(*======================================================================================================================================*)
(*//=============================================================================\\
||  _   _ _  __  _         _                        _   _                      ||
|| | \ | | |/ / / \  _   _| |_ ___  _ __ ___   __ _| |_(_) ___  _ __         ||
|| |  \| | ' / / _ \| | | | __/ _ \| '_ ` _ \ / _` | __| |/ _ \| '_ \        ||
|| | |\  | . \/ ___ \ |_| | || (_) | | | | | | (_| | |_| | (_) | | | |       ||
|| |_| \_|_|\_\_/  \_\__,_|\__\___/|_| |_| |_|\__,_|\__|_|\___/|_| |_|       ||
||                                                                             ||
\\=============================================================================//
fb_RS485FiFoMaster:	Einfaches Senden eines Telegrams über RS485*)
(*
Date          	| Version    	| created under        	| Author          	| Remark *)
(*====================================================================================================================================================*)
(*10/05/2025   	| 1.00      		| TC3		  		| N.Kersting       | first release *)
(*10/05/2025   	| 1.01      		| TC3		  		| N.Kersting       | Nun wird der Empfang auch mit Implementiert  *)
(*13/05/2025   	| 1.02      		| TC3		  		| N.Kersting       | Busbelastungstest Implementiert - Sendet Durchgehend Strings *)
(*14/05/2025   	| 1.03      		| TC3		  		| N.Kersting       | Busauslastung direkt Implementiert *)
(*27/05/2025   	| 1.04      		| TC3		  		| N.Kersting       | Neuen Manuell Mode implementiert um einen Manuell generierten String allein zu Senden *)
(*28/05/2025   	| 1.05      		| TC3		  		| N.Kersting       | Neue Automatisch Ping Funktion hinzugefügt & Wichtiger Bugfix *)
(*02/06/2025   	| 2.00      		| TC3		  		| N.Kersting       | Neue Verbesserte Collision Detection, verhindert, dass Senden bei gefülltem Epmfangspuffer *)
(*03/06/2025   	| 2.01      		| TC3		  		| N.Kersting       | Collision Detection nun aufgeeilt in Empfang und Senden *)
(*03/06/2025   	| 2.02      		| TC3		  		| N.Kersting       | Neue Bus Scan Funktion Implementiert, Scannt alle Teilnehmer Ids im Bus (nur im Manuell Mode verfügbar) *)
(*12/01/2026   	| 2.03      		| TC3		  		| N.Kersting       | Nach dem Pingenkann wieder empfangen werden*)
(*13/01/2026   	| 2.04      		| TC3		  		| N.Kersting       | Ping wird Verzögert zwischen jedem Ping, wenn FiFo gefüllt kann Ping unterbrochen werden*)
(*13/01/2026   	| 2.04      		| TC3		  		| N.Kersting       | Bugfix Step 12 nur speichern wenn ID vorhanden ist!*)
(*09/06/2026   	| 2.05      		| TC3		  		| N.Kersting       | Obergrenze für Max Rows FiFo nun fix auf Globalen Wert *)
(*09/06/2026   	| 2.06      		| TC3		  		| N.Kersting       | Integration I_nMaxDevices*)
(*16/09/2026   	| 2.07      		| TC3		  		| N.Kersting       | Collision Detection eingang*)
(*====================================================================================================================================================*)
FUNCTION_BLOCK fb_RS485FiFoMaster_old
VAR_INPUT
	I_nMaxDevices				:INT := cMaxRowCMDFiFo;
	I_sSendCmdFiFo				:ARRAY[1..cMaxRowCMDFiFo] OF STRING(255);
	I_stDeviceIdent				:ARRAY[1..cMaxRowCMDFiFo] OF ST_HausBus_Ident;	(* Um Zyklisch einzelnt anzupingen *)
	
	I_bAutoPing					:BOOL;												(* Wenn Aktiv wird Zyklisch Automatisch ein Ping gesendet, welcher von den einzelnen Kommunikationsbausteinen ausgewertet werden kann *)
	I_tAutoPingTime				:TIME :=T#10S;										(* Die Intervallzeit, Bis ein Auto Ping gesendet wird *)
	
	I_bUseRXCollisionDetection	:BOOL := TRUE;					(* Aktiviert die Empfangs Kollisions Überprüfung *)
	I_bUseTXCollisionDetection	:BOOL := FALSE;					(* Aktiviert die Sende Kollisions Überprüfung *)
	I_tVerzCollisionDetect		:TIME := T#100MS;
	
	I_bManuellMode				:BOOL := FALSE;
	I_bSearchMode				:BOOL := FALSE;
	I_sSendCmdManuell			:STRING(255);
	I_bSendManuell				:BOOL;
	I_bLogger					:BOOL := FALSE;
	I_bResetLog					:BOOL := FALSE;
	I_bExecute					:BOOL := TRUE;
	I_bBusBelastungstest		:BOOL;
	I_bReset					:BOOL;
	I_sStartZeichen				:BYTE := 16#FD;										(* Startzeichen Präfix *)
	I_sEndZeichen				:BYTE := 16#FE;										(* Endzeichen Suffix *)
	I_pTxBuffer					:POINTER TO ComBuffer; 								(* Zeiger auf TX-Buffer*)
	I_pRxBuffer   				:POINTER TO ComBuffer;  							(* Zeiger auf RX-Buffer*)
END_VAR
VAR_OUTPUT
	Q_bSendDoneFiFo				:ARRAY[1..cMaxRowCMDFiFo] OF BOOL; (*GVL_RS485FiFoSend.bSendDoneFiFo[iFiFoRow]*)
	Q_sReceiveString			:STRING(255);		
	Q_lrBusAuslastung			:LREAL;
	Q_bBusy						:BOOL;
	Q_bDone						:BOOL;
	Q_bError					:BOOL;
	Q_sState					:STRING;
	Q_stStates					:ST_FiFoMaster_State;
END_VAR
VAR
(*==========================================================================================================*)
(* Parameter *)
(*==========================================================================================================*)
	bActivateSend				:BOOL := TRUE;					(* Aktiviert das Senden von Nachrichten *)
	bActivateReceive			:BOOL := TRUE;					(* Aktiviert das Empfangen von Nachrichten *)
	
	bUseRXCollisionDetection	:BOOL := TRUE;					(* Aktiviert die Empfangs Kollisions Überprüfung *)
	bUseTXCollisionDetection	:BOOL := FALSE;					(* Aktiviert die Sende Kollisions Überprüfung *)
	tVerzCollisionDetect		:TIME := T#100MS;				(* Zeit, die zum Empfangen bleibt *)
(*==========================================================================================================*)	
	bRXCollisionDetected		:BOOL;
	bTXCollisionDetected		:BOOL;
	bCollisionFree				:BOOL;	
(*==========================================================================================================*)		
	bFirstCycle					:BOOL := TRUE;
	bStringSend					:BOOL := FALSE;
	bBusBelastungstest			:BOOL := FALSE;
	bBusAuslastung				:BOOL := TRUE;
	bPingStart					:BOOL;
	bBusyMem					:BOOL;
(*==========================================================================================================*)	
	sReceivedMEMString			:STRING(255);
	sReceivedString				:STRING(255);
	sStep						:STRING;
	sString						:STRING(255);
	sStringSend					:STRING(255);
(*==========================================================================================================*)		
	iStep						:INT;
	iStepReceive				:INT;
	iMaxBufferBlocking			:INT := 20;
	icntError					:INT;
	iFiFoRow					:INT := 1;
	icntFiFo					:INT;
	i,h							:INT;
	iStepFiFo					:INT;
	iPingRow					:INT;
(*==========================================================================================================*)		

	tonCollisionFree			:ton;	
	tonTimeout					:ton;
	tonPingIntervall			:ton;
	tonPingVerz					:ton;
	tonSend						:ton;
(*==========================================================================================================*)		
	rTrigSendManuell			:r_Trig;
	rTrigSendSearchMode			:r_trig;
	fbSend     					:SendString255;
	fbReceive   				:ReceiveString255;
	
	fbBusAuslastung				:fb_FilterArray;
	
	fbRS485Search				:fb_RS485IdScan;
	
	fbRS485Logger				:fb_RS485Logger;
	
END_VAR

(*============================================================================================*)
(* Laufzeit fehler *)
tonTimeout(
	PT:=T#1S);
	
(*============================================================================================*)		
(* Collision detection, soll verhinddern, dass nicht gesendet wird, wenn Daten im Empfangsüpuffer sind *)
bUseRXCollisionDetection := I_bUseRXCollisionDetection;
bUseTXCollisionDetection := I_bUseTXCollisionDetection;

(* Receive Collision Dectetion *)
bRXCollisionDetected :=	(I_pRxBuffer^.Count > INT_TO_UINT(iMaxBufferBlocking) 
						OR I_pRxBuffer^.FreeByte < (301 -INT_TO_UINT(iMaxBufferBlocking))
						OR I_pRxBuffer^.blocked
						OR I_pRxBuffer^.Error <> 0
						OR fbReceive.StringReceived
						(*OR sReceivedString <> ''*))
						AND bUseRXCollisionDetection;
						
(* Transmit Collision Detection *)
bTXCollisionDetected :=	(I_pTxBuffer^.Count > INT_TO_UINT(iMaxBufferBlocking) 
						OR I_pTxBuffer^.FreeByte < (301 -INT_TO_UINT(iMaxBufferBlocking))
						OR I_pTxBuffer^.blocked
						OR I_pTxBuffer^.Error <> 0)
						AND bUseTXCollisionDetection;
						
(* Collision Detection Verzögern *)	
tVerzCollisionDetect :=		I_tVerzCollisionDetect;
			
tonCollisionFree(
	IN := 	NOT bRXCollisionDetected
			AND NOT bTXCollisionDetected,
	PT := 	tVerzCollisionDetect,
	Q =>	bCollisionFree);

(*============================================================================================*)	
(* Ping Intervall Timer *)		
tonPingIntervall(
	IN := I_bAutoPing
			AND NOT bPingStart,
	PT := I_tAutoPingTime);

tonPingVerz(
	PT := T#100MS);	
	
(*============================================================================================*)	
(* Busbelastungstest *)	
bBusBelastungstest := I_bBusBelastungstest;
sReceivedMEMString:='';

(*============================================================================================*)	
(* Anzahl der gefüllten FiFo Zeilen *)
icntFiFo := 0;
FOR i := 1 TO cMaxRowCMDFiFo BY 1 DO 
	
	IF i <= I_nMaxDevices
	THEN
		IF (I_sSendCmdFiFo[i]<> '')
		THEN
			icntFiFo := icntFiFo +1;
		END_IF
	END_IF
END_FOR

(*============================================================================================*)	
(* Manuelles Senden *)
rTrigSendManuell(
	CLK := I_bSendManuell);

(*============================================================================================*)
CASE iStepFiFo OF
-1:	sStep := 'FiFo INIT';
	bFirstCycle := FALSE;
	Q_bBusy := FALSE;
	bPingStart := FALSE;
	iFiFoRow := 1;
	iPingRow := 1;
	
	FOR h := 1 TO cMaxRowCMDFiFo BY 1 DO
		IF h <= I_nMaxDevices
		THEN
			Q_bSendDoneFiFo[h] :=TRUE;
		END_IF
	END_FOR
	
	iStepFiFo := 0;

(*============================================================================================*)
0:	sStep := 'Warten, dass FiFo gefüllt wird';
	iFiFoRow := 1;
	
	IF iPingRow <= 0
	THEN
		iPingRow := 1;
	END_IF
	
	bStringSend := FALSE;
	Q_bBusy := FALSE;
	tonPingVerz.IN := FALSE;
		
	(* Wenn die Intervall Zeit abgelaufen ist Ping Start setzen *)
	IF tonPingIntervall.Q
	THEN
		bPingStart := TRUE;
	END_IF
	
	(*IF (icntFiFo > 0
		OR  bBusBelastungstest
		OR I_bManuellMode)
		AND NOT bFirstCycle
		AND NOT bPingStart
		AND bCollisionFree
	THEN
		Q_bBusy := TRUE;
		iStepFiFo := 1;
	ELSIF
		bFirstCycle
	THEN
		iStepFiFo := -1;
	ELSIF
	(* (	*)(bPingStart
		AND NOT bFirstCycle)
		(*OR (bPingStart
		AND iPingRow <> cMaxRS485CMDFiFo))*) (* Es stehen noch Ping befehle aus *)
		AND bCollisionFree
		(*AND icntFiFo =0*)
	THEN
		(*iFiFoRow := iPingRow;*)
		iStepFiFo := 10;	(* Ping senden *)
	END_IF*)
	
	IF bFirstCycle
	THEN
		iStepFiFo := -1;
	ELSE
		IF bCollisionFree
		THEN
			IF icntFiFo > 0
				OR  bBusBelastungstest
				OR I_bManuellMode
			THEN
				Q_bBusy := TRUE;
				iStepFiFo := 1;
			ELSE
				IF bPingStart
					OR iPingRow < I_nMaxDevices	(* Ping wurde unterbrochen *)
				THEN
					IF iPingRow < I_nMaxDevices
					THEN
						iFiFoRow := iPingRow;
					ELSE
						iFiFoRow := 1;
					END_IF
					iStepFiFo := 10;	(* Ping senden *)
				END_IF
			END_IF
		END_IF
	END_IF
	
(*============================================================================================*)	
1:	sStep := 'Prüfen ob STRING in FiFo Zeile gefüllt*';
	
	IF I_bSearchMode
	THEN
		sStep :=fbRS485Search.Q_sState;
	END_IF
	
	(* Manueller Modus *)
	IF I_bManuellMode
	THEN
		(* Prüfen ob in der Zeile etwas steht *)
		IF I_sSendCmdManuell <>''
			AND rTrigSendManuell.Q
			AND NOT I_bSearchMode
		THEN
			IF bCollisionFree
			THEN
				sString :=	I_sSendCmdManuell; 
				bStringSend := TRUE;
				Q_bDone := FALSE;
				Q_bError := FALSE;
				iStepFiFo := iStepFiFo+1;
			END_IF
		END_IF
		(* Prüfen ob in der Zeile etwas steht *)
		IF I_bSearchMode
			AND fbRS485Search.Q_bSend
		THEN
			IF bCollisionFree
			THEN
				sString :=	fbRS485Search.Q_sSearchString; 
				bStringSend := TRUE;
				Q_bDone := FALSE;
				Q_bError := FALSE;
				iStepFiFo := iStepFiFo+1;
			END_IF
		END_IF
	ELSE
		(* Prüfen ob in der ausgewählten Zeile etwas steht *)
		sStringSend :=	I_sSendCmdFiFo[iFiFoRow]; 
		IF I_sSendCmdFiFo[iFiFoRow] = ''
		THEN
			IF iFiFoRow< I_nMaxDevices
			THEN
				iFiFoRow := iFiFoRow+1; (* Nächste Zeile, bis etwas drin Steht *)
			ELSE
				IF bBusBelastungstest
				THEN
					sStringSend :=	CONCAT(F_ToCHR(I_sStartZeichen),'ServiceTOOL-BUSBELASTUNGSTEST-BURSTFIREMODE');
					sStringSend :=	CONCAT(sStringSend,F_ToCHR(I_sEndZeichen));
					(* Senden *)
					
					IF  bCollisionFree
					THEN
						sStep := 'Prüfe ob Senden noch aktiv ist';
						bStringSend := TRUE;
						sString :=	sStringSend;
						Q_bDone := FALSE;
						Q_bError := FALSE;
						iStepFiFo := iStepFiFo+1;
					END_IF
				ELSE
					iStepFiFo := 0;	(* Alle Zeilen Abgearbeitet *)
				END_IF
			END_IF
		ELSE
		(* Senden *)
		Q_bSendDoneFiFo[iFiFoRow] :=FALSE;
		
			IF bCollisionFree
			THEN
				sStep := 'Prüfe ob Senden noch aktiv ist';
				bStringSend := TRUE;
				sString :=	sStringSend;
				Q_bDone := FALSE;
				Q_bError := FALSE;
				iStepFiFo := iStepFiFo+1;
			END_IF
		END_IF
	END_IF
	
(*============================================================================================*)		
2:	sStep := 'Starte Senden';
	Q_bBusy := TRUE;
	tonTimeout.IN := fbSend.Busy;
	
	IF NOT fbSend.Busy
		AND NOT fbReceive.StringReceived
	THEN
		sString := '';
		tonSend.IN := FALSE;
		bStringSend := FALSE;
		iStepFiFo := iStepFiFo+1;
	ELSIF
		(fbSend.Error >0)
		AND NOT (fbSend.Error = 2)
	THEN
		sStep := CONCAT('ERROR-',sStep);
		sStep := CONCAT(sStep,'- ');
		sStep := CONCAT(sStep,INT_TO_STRING(fbSend.Error));
		iStepFiFo := -2;
	ELSIF
		tonTimeout.Q
	THEN
		sStep := CONCAT('ERROR- Timeout',sStep);
		iStepFiFo := -2;
	END_IF
	
(*============================================================================================*)		
3:	(* Senden*)		
	Q_bSendDoneFiFo[iFiFoRow] :=TRUE;
	
	IF iFiFoRow< I_nMaxDevices
		AND NOT I_bSearchMode
	THEN
		iFiFoRow := iFiFoRow+1;
		iStepFiFo := 1;
	ELSE
		Q_bDone := TRUE;
		
		IF (NOT fbRS485Search.Q_bSend
			AND I_bSearchMode)
			OR NOT I_bSearchMode
		THEN
			iStepFiFo := 0;
		END_IF
		
	END_IF
	
(*============================================================================================*)	
(* Ping Senden Ablauf *)
(*============================================================================================*)	
10:	sStep := 'Sende Ping*';
	
	tonPingVerz.IN := FALSE;
	
	(* Ping String erstellen *)
	sStringSend:=	CONCAT(F_ToCHR(I_sStartZeichen),DINT_TO_STRING(I_stDeviceIdent[iFiFoRow].diID));
	sStringSend :=	CONCAT(sStringSend,'.');
	sStringSend :=	CONCAT(sStringSend ,I_stDeviceIdent[iFiFoRow].sPingIdent); 
	sStringSend :=	CONCAT(sStringSend,F_ToCHR(I_sEndZeichen));
	
	IF I_stDeviceIdent[iFiFoRow].sPingIdent = ''
		OR I_stDeviceIdent[iFiFoRow].diID = 0
	THEN
		IF iFiFoRow < I_nMaxDevices
		THEN
			iFiFoRow := iFiFoRow+1; (* Nächste Zeile, bis etwas drin Steht *)
		ELSE
			bPingStart := FALSE;
			iPingRow := I_nMaxDevices;
			iStepFiFo := 0;	(* Alle Zeilen Abgearbeitet *)
		END_IF
	ELSE
	(* Senden *)	
		IF bCollisionFree
		THEN
			sStep := 'Prüfe ob Senden noch aktiv ist';
			bStringSend := TRUE;
			sString :=	sStringSend;
			Q_bDone := FALSE;
			Q_bError := FALSE;
			iStepFiFo := iStepFiFo+1;
		END_IF
	END_IF
	
(*============================================================================================*)		
11:	sStep := 'Starte Senden';
	Q_bBusy := TRUE;
	tonTimeout.IN := fbSend.Busy;
	
	IF NOT fbSend.Busy
		(*AND NOT fbReceive.StringReceived*)
	THEN
		tonSend.IN := FALSE;
		bStringSend := FALSE;
				
		IF NOT fbReceive.StringReceived
			AND bCollisionFree
		THEN
			iStepFiFo := iStepFiFo+1;
		END_IF
		
	ELSIF
		(fbSend.Error >0)
		AND NOT (fbSend.Error = 2)
	THEN
		sStep := CONCAT('ERROR-',sStep);
		sStep := CONCAT(sStep,'- ');
		sStep := CONCAT(sStep,INT_TO_STRING(fbSend.Error));
		iStepFiFo := -2;
	ELSIF
		tonTimeout.Q
	THEN
		sStep := CONCAT('ERROR- Timeout',sStep);
		iStepFiFo := -2;
	END_IF
	
(*============================================================================================*)		
12:	(* Senden*)		
	(* Nur speichern wenn auch wirklich eine ID vorhanden ist *)	
	IF I_stDeviceIdent[iFiFoRow].sPingIdent = ''
		OR I_stDeviceIdent[iFiFoRow].diID = 0
	THEN
		IF iFiFoRow < I_nMaxDevices
		THEN
			iFiFoRow := iFiFoRow+1; (* Nächste Zeile, bis etwas drin Steht *)
		ELSE
			bPingStart := FALSE;
			iPingRow := I_nMaxDevices;
			iStepFiFo := 0;	(* Alle Zeilen Abgearbeitet *)
		END_IF
	ELSE
		IF iFiFoRow < I_nMaxDevices
		THEN
			iFiFoRow := iFiFoRow+1;
			iPingRow := iFiFoRow; (* Zeile speichern *)
			iStepFiFo := 13;	(* Falls das warten Deaktiviert werden soll, kann hier einfach in 10 gesprungen werden *)
		ELSE
			bPingStart := FALSE; (* Letzte Ping Zeile erreicht, Timer zurücksetzen  *)
			iPingRow := I_nMaxDevices;
			iStepFiFo := 13;
		END_IF
	END_IF
(*============================================================================================*)		
13:	(* Optionale Wartezeit zwischen jedem Ping*)		
	tonPingVerz.IN := TRUE;
			
	IF tonPingVerz.Q
	THEN
		IF NOT fbReceive.StringReceived
			AND bCollisionFree
		THEN
			tonPingVerz.IN := FALSE;
			
			IF iFiFoRow < I_nMaxDevices
			THEN
				iStepFiFo := 10; (* nächsten Ping senden *)
			ELSE
				iStepFiFo := 0;
			END_IF
		END_IF
	ELSE
		(* Prüfen ob ein Sendeauftrag anliegt *)
		IF icntFiFo >0
		THEN
			tonPingVerz.IN := FALSE;
			iStepFiFo := 0; (* Sende FiFo leeren *)
		END_IF  
	END_IF
ELSE
(*============================================================================================*)
	Q_bError := TRUE;
	Q_bBusy := FALSE;
	bBusyMem := FALSE;
	tonTimeout.IN := FALSE;
	
	IF I_bReset
	THEN
		iStepFiFo := 0;
	END_IF
END_CASE

(*============================================================================================*)	
(* Nur Senden, wenn nicht Empfangen wird *)
IF bStringSend
THEN
	IF bActivateSend
	THEN
		(* Senden *)
		fbSend(
			SendString:= 	sString,
			TXbuffer:= 		I_pTxBuffer^);
	END_IF
	
ELSE
	IF bActivateReceive
	THEN
		(* Empfangen *)
		ac00_Receive();
	END_IF
END_IF

(*============================================================================================*)	
(* Empfangsmerker 0 Setzen am ende Eines Zyklus *)
Q_sReceiveString := sReceivedMEMString;

(*============================================================================================*)	
(* Busauslastung tracken*)
ac99_Diagnose();

(*============================================================================================*)	
(* StatusStruktur für Visu *)
Q_sState :=	sStep;
Q_stStates.bBusy				:=	Q_bBusy;
Q_stStates.bDone				:=	Q_bDone;
Q_stStates.bError				:=	Q_bError;
Q_stStates.iFiFoCount			:=	icntFiFo;
Q_stStates.iFiFoRow				:=	iFiFoRow;
Q_stStates.lrBusAuslastung		:=	Q_lrBusAuslastung;
Q_stStates.sReceiveString 		:=	Q_sReceiveString;
Q_stStates.sSendString 			:=	sString;
Q_stStates.sState 				:=	Q_sState;

(*============================================================================================*)	
(* RS485 Telegramm Logging *)
fbRS485Logger(
	I_bExecute:= 		I_bLogger,						(* oder eine externe Variable *)
	I_bReset:=			I_bResetLog,	
	I_sTxTelegram:= 	sString,
	I_sRxTelegram:= 	sReceivedMEMString);

ACTION ac00_Receive:
(*============================================================================================*)	
(* Empfangen *)

CASE iStepReceive OF		
0:	fbReceive(
		Prefix := 			F_ToCHR(I_sStartZeichen),
		Suffix := 			F_ToCHR(I_sEndZeichen),
		Timeout:= , 
		Reset:= , 
		StringReceived=> , 
		Busy=> , 
		Error=> , 
		RxTimeout=> , 
		ReceivedString:= 	sReceivedString, 
		RXbuffer:= 			I_pRxBuffer^);
		
	IF fbReceive.StringReceived
	THEN
		iStepReceive := 1;
		sReceivedMEMString := sReceivedString;
	END_IF
	
1:	sReceivedString := '';
	iStepReceive := 0;

	
END_CASE
END_ACTION

ACTION ac99_Diagnose:
(*============================================================================================*)	
(* Busauslastung Prüfen *)

fbBusAuslastung(
	I_bExcecute:= 	bBusAuslastung, 
	I_nWert:= 		UINT_TO_LREAL(I_pTxBuffer^.Count), 
	I_nFilterWert:= 50, 
	Q_nFilter=> 	Q_lrBusAuslastung);
	
	
fbRS485Search(
	I_bStartSearch:= 	I_bSearchMode, 
	I_diStartID:= , 
	I_diMaxID:= , 
	I_sStartZeichen:= 	I_sStartZeichen, 
	I_sEndZeichen:= 	I_sEndZeichen, 
	I_tWait:= , 
	I_StringReceived:= 	sReceivedMEMString, 
	Q_bSend=> , 
	Q_sSearchString=> );
END_ACTION

END_FUNCTION_BLOCK

(* stored: Version 1.1.0.1, ProductVersion 3.1.4024.16
   POU fb_RS485FiFoMaster_old: Id {abb7ee14-f2e6-4645-9657-7cebd7b41d33}, SpecialFunc None
   Action ac00_Receive: Id {c12285ff-9b41-4e09-9783-e6434850ec65}
   Action ac99_Diagnose: Id {729e27f4-8df9-41ab-a478-b2f1a8116421} *)
